TYPE Vec3i : ARRAY[1..3] OF INT; END_TYPE

(* stored: Version 1.1.0.1, ProductVersion 3.1.4024.12
   DUT Vec3i: Id {53fd693e-34e5-49a9-a06b-f11f26280b26} *)
